(* PLC project Generated.project, CODESYS CODESYS V3.5 SP19 Patch 1 *)
(* stored: creationDateTime 2026-09-23T09:52:47.229015, modificationDateTime 2026-09-23T09:52:47.229015 *)

{attribute 'qualified_only'}
{attribute 'strict'}
TYPE E_TranslationFinalInterlockReason : (NONE := 0, BRAKE_COMMAND_NOT_CONFIRMED := 1, RESTART_INHIBITED := 2);
END_TYPE

(* ======================================================================= 🧩 ST_Fault — Brique socle défaut (2 vues : live + latchée) ─────────────────────────────────────────────────────────────── 🎯 Rôle : porter l'état défaut d'un composant, applicable dans TOUS les cas (acquittable ou non), sans brique warning séparée. • Vue LIVE (Error / ErrorId) : suit la cause, retombe seule à 0. • Vue LATCHÉE (Latched / LatchedId): mémorisée au défaut, reste jusqu'au front Reset. Le choix acquittable / non-acquittable se fait PAR CAUSE (ST_FaultCause.Latching), jamais par bloc. 🔒 Sécurité : interlock TOUJOURS sur la cause brute (Error / ErrorId), jamais sur l'acquittement. Reset TOUJOURS effectif, jamais conditionné (std §9). 🧬 Composition : brique de base réutilisable — sortie de FB, struct métier, GVL. Texte IHM NON stocké ici : dérivé côté IHM depuis LatchedId / ErrorId. 📄 Doc : DOC/STDS/CODE_QUALITY_STANDARDS.md §2quinquies / §9 ======================================================================= *)
TYPE ST_Fault : STRUCT
  Error : BOOL;  (* <-- [DIAG] vue LIVE : au moins une cause présente maintenant *)
  ErrorId : WORD;  (* <-- [DIAG] bitfield des causes présentes maintenant (0 si aucune) *)
  Latched : BOOL;  (* <-- [DIAG] vue LATCHÉE : défaut non acquitté, reste jusqu'au front Reset *)
  LatchedId : WORD;  (* <-- [DIAG] ErrorId figé à l'apparition du défaut, effacé au Reset *)
END_STRUCT;
END_TYPE

(* ======================================================================= 🧩 ST_FaultCause — Cause élémentaire alimentant ST_Fault (socle FB_FaultCore) ─────────────────────────────────────────────────────────────── 🎯 Rôle : une cause exprimée EN CLAIR (BOOL + libellé), sans bitfield ni masque. Le FB métier remplit une liste (ARRAY[0..15] OF ST_FaultCause) ; le socle FB_FaultCore en déduit ST_Fault (vue live + vue latchée). 🔒 Sécurité : interlock TOUJOURS sur Active (cause brute), jamais sur le latch. Latching = TRUE → la cause ARME la vue latchée (défaut à acquitter). Latching = FALSE → la cause n'alimente que la vue live (retombe seule). Fail-safe : une cause laissée à Latching=FALSE reste visible en live — pour la rendre acquittable, il faut le déclarer explicitement. 📄 Doc : DOC/STDS/CODE_QUALITY_STANDARDS.md §2quinquies / §9 ======================================================================= *)
TYPE ST_FaultCause : STRUCT
  Active : BOOL;  (* 1 = cause présente maintenant (interlock sur cette valeur) *)
  Latching : BOOL;  (* 1 = cause à acquitter (arme Latched) ; 0 = live seulement *)
  Texte : STRING;  (* libellé prêt IHM (non stocké dans ST_Fault, dérivé côté IHM) *)
END_STRUCT;
END_TYPE

(* ======================================================================= 🛡️ FB_TranslationOutputInterlock — Barrière finale frein / AC600 M3 ─────────────────────────────────────────────────────────────── 🎯 Rôle : Barrière de sécurité finale pour frein et variateur AC600 M3 📄 Doc métier : DOC/AF/AF_Partie-11_Fonction_Translation_v2.3.md 🔌 Interface : Interlock de sortie (entre FB_Translation et PRG_06_Outputs) 🔒 Sécurité : Surveillance feedback frein et watchdog de desserrage ======================================================================= *)
FUNCTION_BLOCK FB_TranslationOutputInterlock
  VAR_INPUT
    Enable : BOOL;  (* === COMMANDES & ETATS GENERAL === --> [CMD] Autorisation generale FB (TRUE=Autorise) *)
    Reset : BOOL;  (* --> [CMD] Acquittement defaut sur front *)
    SafeStop : BOOL;  (* --> [SAFE] Entree securite pour interface standard *)
    PowerContactorEngaged : BOOL;  (* --> [SAFE] Chaine AU rearmee et puissance OK *)
    EffectivePermitM3_Tremie : BOOL;  (* --> [SAFE] Permis Tremie *)
    EffectivePermitM3_Maintenance : BOOL;  (* --> [SAFE] Permis Maintenance *)
    BrakeReleaseRequest : BOOL;  (* === DEMANDES DE COMMANDE AMONT === --> [CMD] Demande de desserrage frein *)
    BrakeCommandOpenConfirmed : BOOL;  (* --> [HW] Confirmation ouverture frein (contacteur/bobine) *)
    RequestedDriveControlWord : WORD;  (* --> [CMD] Mot de commande variateur (0=None, 1=Fwd, 2=Rev, 7=Reset) *)
    RequestedDriveFreqHz : REAL;  (* --> [CMD] Frequence de consigne variateur (Hz) *)
  END_VAR
  VAR_OUTPUT
    Ready : BOOL;  (* === ETATS IEC & SYNOPTIQUE === <-- [STAT] FB pret a fonctionner (sortie libre, hors ST_Status) *)
    Fault : ST_Fault;  (* 🧩 Statut transverse (forme cible ST_Fault) *)
    Reason : E_TranslationFinalInterlockReason;  (* <-- [DIAG] Cause de blocage *)
    DriveControlWord : WORD;  (* === ORDRES ACTIONNEURS VALIDES === <-- [ACT] Mot de commande variateur valide *)
    DriveFreqCmd_Hz : REAL;  (* <-- [ACT] Frequence de consigne variateur valide (Hz) *)
    DriveFreqCmdWord : WORD;  (* <-- [ACT] Frequence mise a l'echelle registre PDO 0x3100 *)
    BrakeCmd : BOOL;  (* <-- [ACT] Ordre ouverture frein valide *)
    BrakeTimeoutElapsed : TIME;  (* === DIAGNOSTICS & TEMPORISATIONS === <-- [DIAG] Ecoule temporisation watchdog frein *)
    RestartInhibit : BOOL;  (* <-- [DIAG] Inhibition redemarrage actif *)
  END_VAR
  VAR
    ResetEdge : R_TRIG;  (* === DETECTEURS DE FRONTS === . [LOC] Detecteur front montant Reset *)
    BrakeTimeoutCauseEdge : R_TRIG;  (* . [LOC] Detecteur nouvelle occurrence cause timeout *)
    BrakeTimeout : TON;  (* === TEMPORISATEURS INTERNES === . [LOC] Temporisateur watchdog desserrage frein *)
    MovementRequested : BOOL;  (* === VARIABLES LOCALES INTERNES === . [LOC] Demande de mouvement active *)
    PermitFinalBlocked : BOOL;  (* . [LOC] Veto directionnel final *)
    NeutralRequestSeen : BOOL;  (* . [LOC] Demande neutre (mot 0) observee *)
    ResetRequired : BOOL;  (* . [LOC] Front Reset obligatoire avant nouvelle marche *)
    BrakeTimeoutCause : BOOL;  (* . [LOC] Cause brute timeout desserrage frein *)
    BrakeTimeoutAck : BOOL := TRUE;  (* . [LOC] Accuse operateur (TRUE = pas d'alarme) *)
    instFault : FB_FaultCore;  (* === SOCLE DEFAUT === * [INST] Socle défaut transverse *)
    instCauses : ARRAY[0..15] OF ST_FaultCause;  (* . [LOC] Table des causes nommées *)
    DriveFreqWordScale : REAL := 100;  (* === ECHELLE & BORNES REGISTRE PDO === Echelle registre 0x3100 (WORD=5000 -> 50,00 Hz) *)
    DriveFreqWordMaxHz : REAL := 600;  (* Borne haute anti-debordement WORD (Hz) *)
  END_VAR

            

// ── 1. FRONT RESET AVANT GATE ───────────────────────────────────────────
ResetEdge(CLK := Reset);

IF NOT Enable OR NOT PowerContactorEngaged THEN
    BrakeTimeout(IN := FALSE, PT := T#500ms);
    DriveControlWord := 0;
    DriveFreqCmd_Hz := 0.0;
    DriveFreqCmdWord := 0;
    BrakeCmd := FALSE;
    BrakeTimeoutElapsed := T#0ms;
    Ready := FALSE;
    Reason := E_TranslationFinalInterlockReason.NONE;
    RETURN;
END_IF;

MovementRequested := (RequestedDriveControlWord = 1) OR (RequestedDriveControlWord = 2);
PermitFinalBlocked := ((RequestedDriveControlWord = 1) AND NOT EffectivePermitM3_Tremie)
                   OR ((RequestedDriveControlWord = 2) AND NOT EffectivePermitM3_Maintenance);

// ── 2. Watchdog : exclusivement après ordre effectif de desserrage ──────
BrakeTimeout(
    IN := BrakeReleaseRequest AND NOT BrakeCommandOpenConfirmed AND NOT RestartInhibit,
    PT := T#500ms
);
BrakeTimeoutElapsed := BrakeTimeout.ET;

IF BrakeTimeout.Q THEN
    BrakeTimeoutCause := TRUE;
ELSIF BrakeCommandOpenConfirmed THEN
    BrakeTimeoutCause := FALSE;
END_IF;

BrakeTimeoutCauseEdge(CLK := BrakeTimeoutCause);
IF BrakeTimeoutCauseEdge.Q THEN
    BrakeTimeoutAck := FALSE;
    RestartInhibit := TRUE;
    ResetRequired := TRUE;
    NeutralRequestSeen := FALSE;
    Reason := E_TranslationFinalInterlockReason.BRAKE_COMMAND_NOT_CONFIRMED;
END_IF;

IF ResetEdge.Q THEN
    BrakeTimeoutAck := TRUE;
    ResetRequired := FALSE;
END_IF;

instCauses[0].Active   := BrakeTimeoutCause OR NOT BrakeTimeoutAck;
instCauses[0].Latching := TRUE;
instCauses[0].Texte    := 'Timeout confirmation ouverture frein translation';

instFault(Enable := Enable, Reset := Reset, Causes := instCauses);
Fault := instFault.Fault;

// ── 3. Réarmement anti-redémarrage automatique ──────────────────────────
IF RestartInhibit AND NOT Fault.Error AND NOT ResetRequired AND NOT ResetEdge.Q THEN
    IF RequestedDriveControlWord = 0 THEN
        NeutralRequestSeen := TRUE;
    ELSIF NeutralRequestSeen AND MovementRequested THEN
        RestartInhibit := FALSE;
        NeutralRequestSeen := FALSE;
    END_IF;
END_IF;

// ── 4. Décision finale : zéro couple utile sans confirmation frein ──────
DriveControlWord := 0;
DriveFreqCmd_Hz := 0.0;
DriveFreqCmdWord := 0;

BrakeCmd := BrakeReleaseRequest AND NOT Fault.Error AND NOT RestartInhibit;
Ready := NOT Fault.Error AND NOT RestartInhibit;

IF RequestedDriveControlWord = 7 THEN
    BrakeCmd := FALSE;
    DriveControlWord := 7;
ELSIF Fault.Error THEN
    BrakeCmd := FALSE;
ELSIF RestartInhibit THEN
    Reason := E_TranslationFinalInterlockReason.RESTART_INHIBITED;
ELSIF MovementRequested AND NOT PermitFinalBlocked THEN
    IF BrakeReleaseRequest AND BrakeCommandOpenConfirmed THEN
        DriveControlWord := RequestedDriveControlWord;
        DriveFreqCmd_Hz := MAX(0.0, RequestedDriveFreqHz);
    END_IF;
END_IF;

// ── 5. Mise à l'échelle finale REAL Hz -> WORD registre PDO 0x3100 ──────
DriveFreqCmdWord := REAL_TO_WORD(LIMIT(0.0, DriveFreqCmd_Hz, DriveFreqWordMaxHz) * DriveFreqWordScale);

          
END_FUNCTION_BLOCK

(* ======================================================================= 🧩 FB_FaultCore — Socle de remplissage de ST_Fault (vue live + vue latchée) ─────────────────────────────────────────────────────────────── 🎯 Rôle : à partir d'une LISTE de causes en clair (ARRAY[0..15] OF ST_FaultCause), produire la brique ST_Fault : • Error / ErrorId : vue LIVE, suit les causes Active, retombe seule. • Latched / LatchedId: vue LATCHÉE, chaque bit figé à l'apparition d'une cause `Active AND Latching`, conservé jusqu'au front Reset. 🔒 Sécurité : - interlock TOUJOURS sur `Causes[i].Active` (cause brute), jamais sur le latch. - Reset TOUJOURS effectif, jamais conditionné (std §9) — agit même Enable=FALSE. - Latching=FALSE → cause visible en LIVE seulement (fail-safe : reste visible). - un défaut laté non acquitté reste publié même FB désactivé (pas d'effacement silencieux sur bascule Enable OFF→ON sans Reset). - une cause à acquitter réapparue re-arme son bit (ré-alarme). 🧬 Un seul socle, réutilisé par tout FB `standard` qui expose un ST_Fault. Pas de State, pas de Warning, pas de texte — hors périmètre de ce socle. 📄 Doc : DOC/STDS/CODE_QUALITY_STANDARDS.md §2quinquies / §9 ======================================================================= *)
FUNCTION_BLOCK FB_FaultCore
  VAR_INPUT
    Enable : BOOL;  (* --> [CMD] Autorisation générale du FB porteur *)
    Reset : BOOL;  (* --> [CMD] Front d'acquittement (jamais conditionné, §9) *)
    Causes : ARRAY[0..15] OF ST_FaultCause;  (* --> [CMD] Liste des causes en clair (Active / Latching / Texte) *)
  END_VAR
  VAR_OUTPUT
    Ready : BOOL;  (* <-- [STAT] FB porteur autorisé (= Enable) *)
    Fault : ST_Fault;  (* <-- [DIAG] Brique défaut (mappée 1:1 sur la sortie du FB porteur) *)
  END_VAR
  VAR
    ResetEdge : R_TRIG;  (* . [LOC] Front montant Reset *)
    Latch : ARRAY[0..15] OF BOOL;  (* . [LOC] Bit laté par cause, jusqu'au Reset *)
    i : INT;  (* . [LOC] Index de parcours de la liste *)
  END_VAR

            

{region "§1 Reset (front, toujours effectif)"}
// Front Reset : efface tous les latches. Jamais conditionné, agit même Enable=FALSE (§9).
Ready := Enable;
ResetEdge(CLK := Reset);
IF ResetEdge.Q THEN
    FOR i := 0 TO 15 DO Latch[i] := FALSE; END_FOR;
END_IF;
{endregion}

{region "§2 Vue LIVE — Error / ErrorId"}
// Bitfield des causes présentes MAINTENANT. Retombe seule à 0 quand les causes disparaissent.
// Non évaluée si Enable=FALSE (pas de lecture de cause hors autorisation).
Fault.ErrorId := 0;
IF Enable THEN
    FOR i := 0 TO 15 DO
        IF Causes[i].Active THEN
            Fault.ErrorId := Fault.ErrorId OR SHL(WORD#1, INT_TO_DWORD(i));
        END_IF;
    END_FOR;
END_IF;
Fault.Error := (Fault.ErrorId <> 0);
{endregion}

{region "§3 Armement des latches (causes à acquitter)"}
// Une cause Active ET Latching arme son bit ; le bit reste jusqu'au front Reset (§1),
// même si la cause disparaît. Réapparition => ré-armement (ré-alarme).
IF Enable THEN
    FOR i := 0 TO 15 DO
        IF Causes[i].Active AND Causes[i].Latching THEN
            Latch[i] := TRUE;
        END_IF;
    END_FOR;
END_IF;
{endregion}

{region "§4 Vue LATCHÉE — Latched / LatchedId"}
// Toujours publiée, y compris Enable=FALSE : un défaut non acquitté reste visible.
Fault.LatchedId := 0;
FOR i := 0 TO 15 DO
    IF Latch[i] THEN
        Fault.LatchedId := Fault.LatchedId OR SHL(WORD#1, INT_TO_DWORD(i));
    END_IF;
END_FOR;
Fault.Latched := (Fault.LatchedId <> 0);
{endregion}

          
END_FUNCTION_BLOCK
